// TwinCAT 3 PLC project TankFuellAnlage
// ProgramVersion: 3.1.4022.1
// libraries:
//   Tc2_Standard, * (Beckhoff Automation GmbH)
//   Tc2_System, * (Beckhoff Automation GmbH)
//   Tc3_Module, * (Beckhoff Automation GmbH)
//   VisuSymbols,3.5.10.0,System
// project tree:
//   / Bildersammlung.TcIPO (not stored), GlobalTextList.TcGTLO, PlcTask.TcTTO (not stored), Visualization Manager.TcVMO (not stored)
//   GVLs/ DIO.TcGVL
//   POUs/ DigitalTwin.TcPOU, MAIN.TcPOU
//   VISUs/ TankFuellAnlage.TcVIS
// real-time tasks:
//   TASK PlcTask: cycle T#10ms, priority 20, ADS port 350
// motion (NC):
//   TASK NC-Task 1 SAF: cycle T#2ms, priority 4, ADS port 501
//   TASK NC-Task 1 SVB: cycle T#10ms, priority 8, ADS port 511
//   AXIS Axis 1 (id 1)
//     OtherSettings: AllowMotionCmdToSlave=true
//     encoder EncType=4
//       EncPara: MaxCount=#x0000ffff
//         Inc: RefSoftSyncMask=#x0000ffff
//     drive DrvType=24
//       Analog: ScaleFactorActTorque=0.1
//       TimeComp: TaskDelayCycles=1
//     controller CtrType=1
//       CtrPara: PriorControlFactor=1
//         Observer: BandWidth=20
//   AXIS Axis 2 (id 2)
//     OtherSettings: AllowMotionCmdToSlave=true
//     encoder EncType=4
//       EncPara: MaxCount=#x0000ffff
//         Inc: RefSoftSyncMask=#x0000ffff
//     drive DrvType=24
//       Analog: ScaleFactorActTorque=0.1
//       TimeComp: TaskDelayCycles=1
//     controller CtrType=1
//       CtrPara: PriorControlFactor=1
//         Observer: BandWidth=20
//   AXIS Axis 3 (id 3)
//     OtherSettings: AllowMotionCmdToSlave=true
//     encoder EncType=4
//       EncPara: MaxCount=#x0000ffff
//     drive DrvType=23
//       Analog: ScaleFactorActTorque=0.1
//       TimeComp: TaskDelayCycles=1
//     controller CtrType=1
//       CtrPara: PriorControlFactor=1
//         Observer: BandWidth=20
//   AXIS Axis 4 (id 4)
//     OtherSettings: AllowMotionCmdToSlave=true
//     encoder EncType=4
//       EncPara: MaxCount=#x0000ffff
//     drive DrvType=23
//       Analog: ScaleFactorActTorque=0.1
//       TimeComp: TaskDelayCycles=1
//     controller CtrType=1
//       CtrPara: PriorControlFactor=1
//         Observer: BandWidth=20
//   AXIS Axis 5 (id 5)
//     OtherSettings: AllowMotionCmdToSlave=true
//     encoder EncType=19
//       EncPara: MaxCount=#xffffffff
//     drive DrvType=16
//       DrvPara: MaxCount=#xffffffff
//         Analog: ScaleFactorActTorque=0.1
//         TimeComp: TaskDelayCycles=1
//     controller CtrType=1
//       CtrPara: PriorControlFactor=1
//         Observer: BandWidth=20
//   AXIS Axis 6 (id 6)
//     OtherSettings: AllowMotionCmdToSlave=true
//     encoder EncType=19
//       EncPara: MaxCount=#xffffffff
//     drive DrvType=16
//       DrvPara: MaxCount=#xffffffff
//         Analog: ScaleFactorActTorque=0.1
//         TimeComp: TaskDelayCycles=1
//     controller CtrType=1
//       CtrPara: PriorControlFactor=1
//         Observer: BandWidth=20
// I/O:
//   DEVICE Device 1 (EtherCAT), AmsNetId 5.35.139.20.2.1
//     Term 1 (EK1200) [EK1200-5000 EtherCAT Power supply (2A E-Bus)]
//       Term 2 (EL1809) [EL1809 16Ch. Dig. Input 24V, 3ms]
//       Term 3 (EL1809) [EL1809 16Ch. Dig. Input 24V, 3ms]
//       Term 4 (EL2809) [EL2809 16Ch. Dig. Output 24V, 0.5A]
//       Term 5 (EL2809) [EL2809 16Ch. Dig. Output 24V, 0.5A]
//       Term 6 (EL3064) [EL3064 4Ch. Ana. Input 0-10V]
//       Term 7 (EL4034) [EL4034 4Ch. Ana. Output +/-10V, 12bit]
//       Term 8 (EL7031) [EL7031 1Ch. Stepper motor output stage (24V, 1.5A)]
//       Term 9 (EL7031) [EL7031 1Ch. Stepper motor output stage (24V, 1.5A)]
//       Term 10 (EL7332) [EL7332 2Ch. DC motor output stage (24V, 1.5A)]
//       Term 11 (EL7201-0010) [EL7201-0010 1Ch. MDP742 Servo motor output stage with OCT (50V, 4A)]
//       Term 12 (EL7201-0010) [EL7201-0010 1Ch. MDP742 Servo motor output stage with OCT (50V, 4A)]
//       Term 26 (EL6090) [EL6090 Display terminal]
//       Term 27 (EK1110) [EK1110 EtherCAT extension]
// variable links:
//   NC-Task 1 SAF/Axes/Axis 1 <-> Device 1 (EtherCAT)/Term 1 (EK1200)/Term 8 (EL7031)
//     Drive/Inputs/In/nState1 @bit 3 <-> STM Status/Status/Error
//     Drive/Inputs/In/nState1 @bit 5 <-> STM Status/Status/Moving negative
//     Drive/Inputs/In/nState1 @bit 4 <-> STM Status/Status/Moving positive
//     Drive/Inputs/In/nState1 @bit 1 <-> STM Status/Status/Ready
//     Drive/Inputs/In/nState1 <-> STM Status/Status/Ready to enable
//     Drive/Inputs/In/nState1 @bit 6 <-> STM Status/Status/Torque reduced
//     Drive/Inputs/In/nState1 @bit 2 <-> STM Status/Status/Warning
//     Drive/Inputs/In/nState2 @bit 3 <-> STM Status/Status/Digital input 1
//     Drive/Inputs/In/nState2 @bit 4 <-> STM Status/Status/Digital input 2
//     Drive/Inputs/In/nState2 @bit 5 <-> STM Status/Status/Sync error
//     Drive/Inputs/In/nState2 @bit 7 <-> STM Status/Status/TxPDO Toggle
//     Drive/Inputs/In/nState4 @bit 1 <-> WcState/InputToggle
//     Drive/Inputs/In/nState4 <-> WcState/WcState
//     Drive/Outputs/Out/nCtrl1 <-> STM Control/Control/Enable
//     Drive/Outputs/Out/nCtrl1 @bit 2 <-> STM Control/Control/Reduce torque
//     Drive/Outputs/Out/nCtrl1 @bit 1 <-> STM Control/Control/Reset
//     Drive/Outputs/Out/nDataOut2[0] <-> STM Velocity/Velocity
//     Enc/Inputs/In/nDataIn1[0] <-> ENC Status compact/Counter value
//     Enc/Inputs/In/nDataIn2[0] <-> ENC Status compact/Latch value
//     Enc/Inputs/In/nState1 @bit 4 <-> ENC Status compact/Status/Counter overflow
//     Enc/Inputs/In/nState1 @bit 3 <-> ENC Status compact/Status/Counter underflow
//     Enc/Inputs/In/nState1 @bit 1 <-> ENC Status compact/Status/Latch extern valid
//     Enc/Inputs/In/nState1 @bit 2 <-> ENC Status compact/Status/Set counter done
//     Enc/Inputs/In/nState2 @bit 4 <-> ENC Status compact/Status/Status of extern latch
//     Enc/Inputs/In/nState2 @bit 5 <-> ENC Status compact/Status/Sync error
//     Enc/Inputs/In/nState2 @bit 7 <-> ENC Status compact/Status/TxPDO Toggle
//     Enc/Inputs/In/nState4 @bit 1 <-> WcState/InputToggle
//     Enc/Inputs/In/nState4 <-> WcState/WcState
//     Enc/Outputs/Out/nCtrl1 @bit 3 <-> ENC Control compact/Control/Enable latch extern on negative edge
//     Enc/Outputs/Out/nCtrl1 @bit 1 <-> ENC Control compact/Control/Enable latch extern on positive edge
//     Enc/Outputs/Out/nCtrl1 @bit 2 <-> ENC Control compact/Control/Set counter
//     Enc/Outputs/Out/nDataOut1[0] <-> ENC Control compact/Set counter value
//   NC-Task 1 SAF/Axes/Axis 2 <-> Device 1 (EtherCAT)/Term 1 (EK1200)/Term 9 (EL7031)
//     Drive/Inputs/In/nState1 @bit 3 <-> STM Status/Status/Error
//     Drive/Inputs/In/nState1 @bit 5 <-> STM Status/Status/Moving negative
//     Drive/Inputs/In/nState1 @bit 4 <-> STM Status/Status/Moving positive
//     Drive/Inputs/In/nState1 @bit 1 <-> STM Status/Status/Ready
//     Drive/Inputs/In/nState1 <-> STM Status/Status/Ready to enable
//     Drive/Inputs/In/nState1 @bit 6 <-> STM Status/Status/Torque reduced
//     Drive/Inputs/In/nState1 @bit 2 <-> STM Status/Status/Warning
//     Drive/Inputs/In/nState2 @bit 3 <-> STM Status/Status/Digital input 1
//     Drive/Inputs/In/nState2 @bit 4 <-> STM Status/Status/Digital input 2
//     Drive/Inputs/In/nState2 @bit 5 <-> STM Status/Status/Sync error
//     Drive/Inputs/In/nState2 @bit 7 <-> STM Status/Status/TxPDO Toggle
//     Drive/Inputs/In/nState4 @bit 1 <-> WcState/InputToggle
//     Drive/Inputs/In/nState4 <-> WcState/WcState
//     Drive/Outputs/Out/nCtrl1 <-> STM Control/Control/Enable
//     Drive/Outputs/Out/nCtrl1 @bit 2 <-> STM Control/Control/Reduce torque
//     Drive/Outputs/Out/nCtrl1 @bit 1 <-> STM Control/Control/Reset
//     Drive/Outputs/Out/nDataOut2[0] <-> STM Velocity/Velocity
//     Enc/Inputs/In/nDataIn1[0] <-> ENC Status compact/Counter value
//     Enc/Inputs/In/nDataIn2[0] <-> ENC Status compact/Latch value
//     Enc/Inputs/In/nState1 @bit 4 <-> ENC Status compact/Status/Counter overflow
//     Enc/Inputs/In/nState1 @bit 3 <-> ENC Status compact/Status/Counter underflow
//     Enc/Inputs/In/nState1 @bit 1 <-> ENC Status compact/Status/Latch extern valid
//     Enc/Inputs/In/nState1 @bit 2 <-> ENC Status compact/Status/Set counter done
//     Enc/Inputs/In/nState2 @bit 4 <-> ENC Status compact/Status/Status of extern latch
//     Enc/Inputs/In/nState2 @bit 5 <-> ENC Status compact/Status/Sync error
//     Enc/Inputs/In/nState2 @bit 7 <-> ENC Status compact/Status/TxPDO Toggle
//     Enc/Inputs/In/nState4 @bit 1 <-> WcState/InputToggle
//     Enc/Inputs/In/nState4 <-> WcState/WcState
//     Enc/Outputs/Out/nCtrl1 @bit 3 <-> ENC Control compact/Control/Enable latch extern on negative edge
//     Enc/Outputs/Out/nCtrl1 @bit 1 <-> ENC Control compact/Control/Enable latch extern on positive edge
//     Enc/Outputs/Out/nCtrl1 @bit 2 <-> ENC Control compact/Control/Set counter
//     Enc/Outputs/Out/nDataOut1[0] <-> ENC Control compact/Set counter value
//   NC-Task 1 SAF/Axes/Axis 3 <-> Device 1 (EtherCAT)/Term 1 (EK1200)/Term 10 (EL7332)
//     Drive/Inputs/In/nState1 @bit 3 <-> DCM Status Channel 1/Status/Error
//     Drive/Inputs/In/nState1 @bit 5 <-> DCM Status Channel 1/Status/Moving negative
//     Drive/Inputs/In/nState1 @bit 4 <-> DCM Status Channel 1/Status/Moving positive
//     Drive/Inputs/In/nState1 @bit 1 <-> DCM Status Channel 1/Status/Ready
//     Drive/Inputs/In/nState1 <-> DCM Status Channel 1/Status/Ready to enable
//     Drive/Inputs/In/nState1 @bit 6 <-> DCM Status Channel 1/Status/Torque reduced
//     Drive/Inputs/In/nState1 @bit 2 <-> DCM Status Channel 1/Status/Warning
//     Drive/Inputs/In/nState2 @bit 3 <-> DCM Status Channel 1/Status/Digital input 1
//     Drive/Inputs/In/nState2 @bit 4 <-> DCM Status Channel 1/Status/Digital input 2
//     Drive/Inputs/In/nState2 @bit 5 <-> DCM Status Channel 1/Status/Sync error
//     Drive/Inputs/In/nState2 @bit 7 <-> DCM Status Channel 1/Status/TxPDO Toggle
//     Drive/Inputs/In/nState4 @bit 1 <-> WcState/InputToggle
//     Drive/Inputs/In/nState4 <-> WcState/WcState
//     Drive/Outputs/Out/nCtrl1 <-> DCM Control Channel 1/Control/Enable
//     Drive/Outputs/Out/nCtrl1 @bit 2 <-> DCM Control Channel 1/Control/Reduce torque
//     Drive/Outputs/Out/nCtrl1 @bit 1 <-> DCM Control Channel 1/Control/Reset
//     Drive/Outputs/Out/nDataOut2[0] <-> DCM Velocity Channel 1/Velocity
//   NC-Task 1 SAF/Axes/Axis 4 <-> Device 1 (EtherCAT)/Term 1 (EK1200)/Term 10 (EL7332)
//     Drive/Inputs/In/nState1 @bit 3 <-> DCM Status Channel 2/Status/Error
//     Drive/Inputs/In/nState1 @bit 5 <-> DCM Status Channel 2/Status/Moving negative
//     Drive/Inputs/In/nState1 @bit 4 <-> DCM Status Channel 2/Status/Moving positive
//     Drive/Inputs/In/nState1 @bit 1 <-> DCM Status Channel 2/Status/Ready
//     Drive/Inputs/In/nState1 <-> DCM Status Channel 2/Status/Ready to enable
//     Drive/Inputs/In/nState1 @bit 6 <-> DCM Status Channel 2/Status/Torque reduced
//     Drive/Inputs/In/nState1 @bit 2 <-> DCM Status Channel 2/Status/Warning
//     Drive/Inputs/In/nState2 @bit 3 <-> DCM Status Channel 2/Status/Digital input 1
//     Drive/Inputs/In/nState2 @bit 4 <-> DCM Status Channel 2/Status/Digital input 2
//     Drive/Inputs/In/nState2 @bit 5 <-> DCM Status Channel 2/Status/Sync error
//     Drive/Inputs/In/nState2 @bit 7 <-> DCM Status Channel 2/Status/TxPDO Toggle
//     Drive/Inputs/In/nState4 @bit 1 <-> WcState/InputToggle
//     Drive/Inputs/In/nState4 <-> WcState/WcState
//     Drive/Outputs/Out/nCtrl1 <-> DCM Control Channel 2/Control/Enable
//     Drive/Outputs/Out/nCtrl1 @bit 2 <-> DCM Control Channel 2/Control/Reduce torque
//     Drive/Outputs/Out/nCtrl1 @bit 1 <-> DCM Control Channel 2/Control/Reset
//     Drive/Outputs/Out/nDataOut2[0] <-> DCM Velocity Channel 2/Velocity
//   NC-Task 1 SAF/Axes/Axis 5 <-> Device 1 (EtherCAT)/Term 1 (EK1200)/Term 11 (EL7201-0010)
//     Drive/Inputs/In/nDcOutputTime <-> InfoData/DcOutputShift
//     Drive/Inputs/In/nState1 <-> DRV Statusword/Statusword
//     Drive/Inputs/In/nState2 <-> DRV Statusword/Statusword @bit 8
//     Drive/Inputs/In/nState4 @bit 1 <-> WcState/InputToggle
//     Drive/Inputs/In/nState4 <-> WcState/WcState
//     Drive/Outputs/Out/nCtrl1 <-> DRV Controlword/Controlword
//     Drive/Outputs/Out/nCtrl2 <-> DRV Controlword/Controlword @bit 8
//     Drive/Outputs/Out/nDataOut2 <-> DRV Target velocity/Target velocity
//     Enc/Inputs/In/nDataIn1 <-> FB Position/Position
//     Enc/Inputs/In/nDcInputTime <-> InfoData/DcInputShift
//     Enc/Inputs/In/nState4 @bit 1 <-> WcState/InputToggle
//     Enc/Inputs/In/nState4 <-> WcState/WcState
//   NC-Task 1 SAF/Axes/Axis 6 <-> Device 1 (EtherCAT)/Term 1 (EK1200)/Term 12 (EL7201-0010)
//     Drive/Inputs/In/nDcOutputTime <-> InfoData/DcOutputShift
//     Drive/Inputs/In/nState1 <-> DRV Statusword/Statusword
//     Drive/Inputs/In/nState2 <-> DRV Statusword/Statusword @bit 8
//     Drive/Inputs/In/nState4 @bit 1 <-> WcState/InputToggle
//     Drive/Inputs/In/nState4 <-> WcState/WcState
//     Drive/Outputs/Out/nCtrl1 <-> DRV Controlword/Controlword
//     Drive/Outputs/Out/nCtrl2 <-> DRV Controlword/Controlword @bit 8
//     Drive/Outputs/Out/nDataOut2 <-> DRV Target velocity/Target velocity
//     Enc/Inputs/In/nDataIn1 <-> FB Position/Position
//     Enc/Inputs/In/nDcInputTime <-> InfoData/DcInputShift
//     Enc/Inputs/In/nState4 @bit 1 <-> WcState/InputToggle
//     Enc/Inputs/In/nState4 <-> WcState/WcState
//   TankFuellAnlage/TankFuellAnlage Instance <-> Device 1 (EtherCAT)/Term 1 (EK1200)/Term 2 (EL1809)
//     PlcTask Inputs/DIO.Stoermeldung <-> Channel 4/Input
//     PlcTask Inputs/DIO.Ventil_1 <-> Channel 1/Input
//     PlcTask Inputs/DIO.Ventil_2 <-> Channel 2/Input
//     PlcTask Inputs/DIO.Ventil_3 <-> Channel 3/Input
//   TankFuellAnlage/TankFuellAnlage Instance <-> Device 1 (EtherCAT)/Term 1 (EK1200)/Term 4 (EL2809)
//     PlcTask Outputs/DIO.Schwimmerschalter_B{1..6} <-> Channel {1..6}/Output  (6 links)

// ---- GVLs/DIO.TcGVL
{attribute 'qualified_only'}
VAR_GLOBAL
	// Digitaler Twin --> Ausgänge der Regelung gehen hier auf Eingänge
	
	Ventil_1 AT %I*: BOOL;
	Ventil_2 AT %I*: BOOL;
	Ventil_3 AT %I*: BOOL;
	Stoermeldung AT %I*:BOOL;
	
	Schwimmerschalter_B1 AT %Q*:BOOL;
	Schwimmerschalter_B2 AT %Q*:BOOL;
	Schwimmerschalter_B3 AT %Q*:BOOL;
	Schwimmerschalter_B4 AT %Q*:BOOL;
	Schwimmerschalter_B5 AT %Q*:BOOL;
	Schwimmerschalter_B6 AT %Q*:BOOL;

END_VAR

// ---- POUs/DigitalTwin.TcPOU
FUNCTION_BLOCK DigitalTwin
VAR_INPUT
END_VAR
VAR_OUTPUT
END_VAR
VAR
	tonTaktgeber: ton;	

	xAuslass1: BOOL;	//Es wird Wasser abgelassen
	xAuslass2: BOOL;
	xAuslass3: BOOL;

	xSchnellEntleeren1:BOOL;
	xSchnellEntleeren2:BOOL;
	xSchnellEntleeren3:BOOL;
	
	uiFuellstandTank1: UINT;	// 0 --> voll; 300 --> leer
	uiFuellstandTank2: UINT;
	uiFuellstandTank3: UINT;	
END_VAR

//Simulation für die Visualisierung
tonTaktgeber(IN:= NOT tonTaktgeber.Q, PT:= T#30MS);


////////////////////////////////////////////
// Achtung: 
//		Füllstand 0 --> Voll
// 		Füllstand 300 --> Leer
//
////////////////////////////////////////////


IF tonTaktgeber.Q THEN
	// damit das Simulation mit passabler Geschwindigkeit läuft	

	// Tank leeren
	IF  xAuslass1 THEN
		IF uiFuellstandTank1 < 300 THEN
			uiFuellstandTank1 := uiFuellstandTank1 + 1;
		ELSE
			uiFuellstandTank1 := 300;		
		END_IF
	END_IF

	IF  xAuslass2 THEN
		IF uiFuellstandTank2 < 300 THEN
			uiFuellstandTank2 := uiFuellstandTank2 + 1;
		ELSE
			uiFuellstandTank2 := 300;		
		END_IF
	END_IF

	IF  xAuslass3 THEN
		IF uiFuellstandTank3 < 300 THEN
			uiFuellstandTank3 := uiFuellstandTank3 + 1;
		ELSE
			uiFuellstandTank3 := 300;		
		END_IF
	END_IF
	
	
	// Tank schnell entleeren
	
	IF  xSchnellEntleeren1 THEN
		IF uiFuellstandTank1 < 290 THEN
			uiFuellstandTank1 := uiFuellstandTank1 + 10;
		ELSE
			uiFuellstandTank1 := 300;		
		END_IF
	END_IF

	IF  xSchnellEntleeren2 THEN
		IF uiFuellstandTank2 < 290 THEN
			uiFuellstandTank2 := uiFuellstandTank2 + 10;
		ELSE
			uiFuellstandTank2 := 300;		
		END_IF
	END_IF

	IF  xSchnellEntleeren3 THEN
		IF uiFuellstandTank3 < 290 THEN
			uiFuellstandTank3 := uiFuellstandTank3 + 10;
		ELSE
			uiFuellstandTank3 := 300;		
		END_IF
	END_IF
	
	
	// Tank füllen
	IF DIO.Ventil_1 THEN
		IF uiFuellstandTank1 > 1 THEN
			uiFuellstandTank1 := uiFuellstandTank1 - 1;
		ELSE
			uiFuellstandTank1 := 0;	
		END_IF
	END_IF
	
	IF DIO.Ventil_2 THEN
		IF uiFuellstandTank2 > 1 THEN
			uiFuellstandTank2 := uiFuellstandTank2 - 1;
		ELSE
			uiFuellstandTank2 := 0;	
		END_IF
	END_IF
	
	IF DIO.Ventil_3 THEN
		IF uiFuellstandTank3 > 1 THEN
			uiFuellstandTank3 := uiFuellstandTank3 - 1;
		ELSE
			uiFuellstandTank3 := 0;	
		END_IF
	END_IF
	
END_IF

////////////////////////////////////////////
// Achtung: 
//		Füllstand 0 --> Voll
// 		Füllstand 300 --> Leer
//
////////////////////////////////////////////


// Füllstand unten
IF uiFuellstandTank1 < 290 THEN
	dio.Schwimmerschalter_B1 := TRUE;
ELSE
	dio.Schwimmerschalter_B1 := FALSE;
END_IF

IF uiFuellstandTank2 < 290 THEN
	dio.Schwimmerschalter_B3 := TRUE;
ELSE
	dio.Schwimmerschalter_B3 := FALSE;
END_IF

IF uiFuellstandTank3 < 290 THEN
	dio.Schwimmerschalter_B5 := TRUE;
ELSE
	dio.Schwimmerschalter_B5 := FALSE;
END_IF


// Füllstand oben
IF uiFuellstandTank1 < 10 THEN
	dio.Schwimmerschalter_B2 := TRUE;
ELSE
	dio.Schwimmerschalter_B2 := FALSE;
END_IF

IF uiFuellstandTank2 < 10 THEN
	dio.Schwimmerschalter_B4 := TRUE;
ELSE
	dio.Schwimmerschalter_B4 := FALSE;
END_IF

IF uiFuellstandTank3 < 10 THEN
	dio.Schwimmerschalter_B6 := TRUE;
ELSE
	dio.Schwimmerschalter_B6 := FALSE;
END_IF

END_FUNCTION_BLOCK

// ---- POUs/MAIN.TcPOU
PROGRAM MAIN
VAR
	DigitalTwin: DigitalTwin;
END_VAR

DigitalTwin();

END_PROGRAM

// ---- GlobalTextList.TcGTLO
TEXTLIST GlobalTextList
  410 = '-B1'
  235 = '-B2'
  26 = '-B3'
  878 = '-B4'
  946 = '-B5'
  390 = '-B6'
  88 = '-Q1'
  726 = '-Q2'
  710 = '-Q3'
  546 = '-Y1'
  973 = 'Auslass'
  141 = 'B2'
  787 = 'Entleeren'
  775 = 'Leeren'
  136 = 'Lüfter 1'
  438 = 'Lüfter 2'
  522 = 'Lüfter 3'
  25 = 'Lüfter 4'
  879 = 'Schnell Entleeren'
  958 = 'Tank 1'
  630 = 'Tank 2'
  349 = 'Tank 3'
  743 = 'Tankfüllanalge - Beispiel 111'
  842 = 'Tankfüllanlage - Beispiel 111'
END_TEXTLIST

// ---- VISUs/TankFuellAnlage.TcVIS
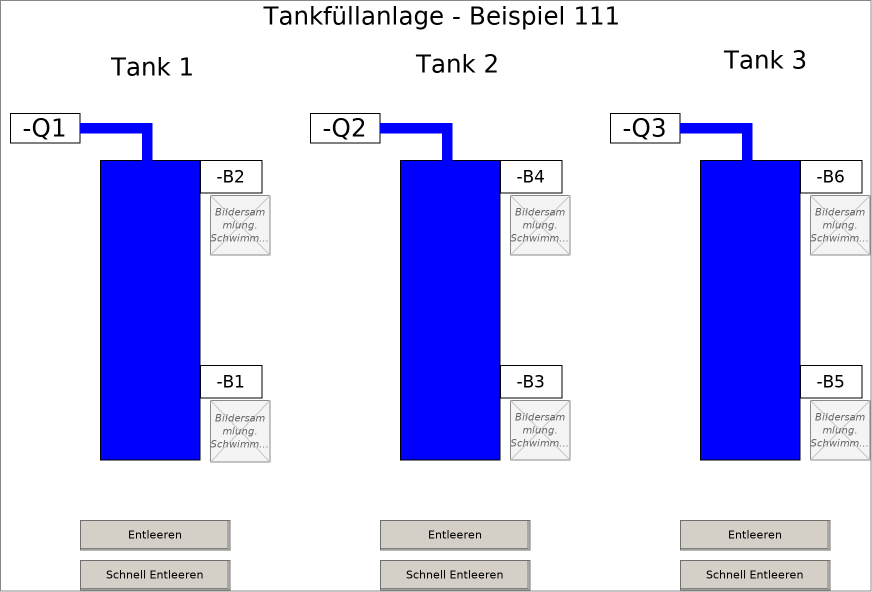
VISUALIZATION TankFuellAnlage  // 872x592
    Polygon (680,123) (752,123) (753,459) (743,459) (742,133) (680,133)
    Polygon (380,123) (452,123) (453,459) (443,459) (442,133) (380,133)
    Polygon (80,123) (152,123) (153,459) (143,459) (142,133) (80,133)
    Rectangle (100,160 100x300)
    Rectangle (100,160 100x300)
        p2773130477: MAIN.DigitalTwin.uiFuellstandTank1
    Label (105,52 95x30), "Tank 1"
    Button (80,520 150x30), "Entleeren"
        tap MAIN.DigitalTwin.xAuslass1
    Rectangle (10,113 70x30), "-Q1", colour toggle: DIO.Ventil_1
    Rectangle (400,160 100x300)
    Rectangle (400,160 100x300)
        p2773130477: MAIN.DigitalTwin.uiFuellstandTank2
    Label (410,49 95x30), "Tank 2"
    Button (380,520 150x30), "Entleeren"
        tap MAIN.DigitalTwin.xAuslass2
    Rectangle (310,113 70x30), "-Q2", colour toggle: DIO.Ventil_2
    Rectangle (391,183 29x301), colour toggle: DIO.Ventil_1
    Rectangle (700,160 100x300)
    Rectangle (700,160 100x300)
        p2773130477: MAIN.DigitalTwin.uiFuellstandTank3
    Label (718,45 95x30), "Tank 3"
    Button (680,520 150x30), "Entleeren"
        tap MAIN.DigitalTwin.xAuslass3
    Rectangle (610,113 70x30), "-Q3", colour toggle: DIO.Ventil_3
    Image (810,195 50x60), invisible if: dio.Schwimmerschalter_B6, image: Bildersammlung.Schwimmerschalter_Offen
    Image (810,195 60x60), invisible if: NOT dio.Schwimmerschalter_B6, image: Bildersammlung.Schwimmerschalter_Betätigt
    Image (810,400 50x60), invisible if: dio.Schwimmerschalter_B5, image: Bildersammlung.Schwimmerschalter_Offen
    Image (510,195 50x60), invisible if: dio.Schwimmerschalter_B4, image: Bildersammlung.Schwimmerschalter_Offen
    Image (510,400 50x60), invisible if: dio.Schwimmerschalter_B3, image: Bildersammlung.Schwimmerschalter_Offen
    Image (210,195 50x60), invisible if: dio.Schwimmerschalter_B2, image: Bildersammlung.Schwimmerschalter_Offen
    Image (210,400 50x60), invisible if: dio.Schwimmerschalter_B1, image: Bildersammlung.Schwimmerschalter_Offen
    Image (810,400 60x60), invisible if: NOT dio.Schwimmerschalter_B5, image: Bildersammlung.Schwimmerschalter_Betätigt
    Image (510,195 60x60), invisible if: NOT dio.Schwimmerschalter_B4, image: Bildersammlung.Schwimmerschalter_Betätigt
    Image (510,400 60x60), invisible if: NOT dio.Schwimmerschalter_B3, image: Bildersammlung.Schwimmerschalter_Betätigt
    Image (210,195 60x60), invisible if: NOT dio.Schwimmerschalter_B2, image: Bildersammlung.Schwimmerschalter_Betätigt
    Image (210,400 60x62), invisible if: NOT dio.Schwimmerschalter_B1, image: Bildersammlung.Schwimmerschalter_Betätigt
    Rectangle (500,160 62x33), "-B4"
    Rectangle (200,160 62x33), "-B2"
    Rectangle (800,160 62x33), "-B6"
    Rectangle (200,365 62x33), "-B1"
    Rectangle (500,365 62x33), "-B3"
    Rectangle (800,365 62x33), "-B5"
    Polygon (80,123) (152,123) (153,459) (143,459) (142,133) (80,133), invisible if: NOT DIO.Ventil_1
    Polygon (380,123) (452,123) (453,459) (443,459) (442,133) (380,133), invisible if: NOT DIO.Ventil_2
    Polygon (680,123) (752,123) (753,459) (743,459) (742,133) (680,133), invisible if: NOT DIO.Ventil_3
    Label (139,1 606x30), "Tankfüllanlage - Beispiel 111"
    Button (80,560 150x30), "Schnell Entleeren"
        tap MAIN.DigitalTwin.xSchnellEntleeren1
    Button (380,560 150x30), "Schnell Entleeren"
        tap MAIN.DigitalTwin.xSchnellEntleeren2
    Button (680,560 150x30), "Schnell Entleeren"
        tap MAIN.DigitalTwin.xSchnellEntleeren3
END_VISUALIZATION
